// TIA Portal V17 export
// export: Created 2023-12-22T15:05:25.2235005Z, ExportSetting WithDefaults, DisplayName Totally Integrated Automation Portal, DisplayVersion V17, DisplayName TIA Portal Openness, DisplayVersion V17, DisplayName TIA Portal Version Control Interface, DisplayVersion V17, DisplayName STEP 7 Professional, DisplayVersion V17, DisplayName STEP 7 Safety, DisplayVersion V17, DisplayName WinCC Advanced, DisplayVersion V17
FUNCTION_BLOCK "Line_Control"   // FB5, LAD
{ S7_Optimized_Access := 'FALSE' }
VERSION : 0.1
// stored: AutoNumber false, IsIECCheckEnabled false, SetENOAutomatically false, UDAEnableTagReadback false
   VAR DB_SPECIFIC
      Local : Bool;   // Локальный
      RESET_STAT : Bool;   // Обнуление статистики за неделю
      Line_Settings : Bool;   // Параметры линии
      Line_Alarms : Bool;   // Аварии линии
      Group1_PolyMix_1 : Bool;   // Группа 1 PolyMix 1
      Group1_PolyMix_2 : Bool;   // Группа 1 PolyMix 2
      Group2_PolyMix_1 : Bool;   // Группа 2 PolyMix 1
      Group2_PolyMix_2 : Bool;   // Группа 2 PolyMix 2
      ALLS : Bool;   // Нижний аварийный уровень
      REQ_Z6_BK1 : Bool;   // Запрос открытия задвижки 6 с БК 1
      REQ_Z6_BK2 : Bool;   // Запрос открытия задвижки 6 с БК 2
      REQ_Z5_Start_A : Bool;   // Запрос открытия задвижки 5
      REQ_Z4_Start_A : Bool;   // Запрос открытия задвижки 4
      REQ_Z3_Start_A : Bool;   // Запрос открытия задвижки 3
      REQ_Z2_Start_A : Bool;   // Запрос открытия задвижки 2
      REQ_Z1_Start_A : Bool;   // Запрос открытия задвижки 1
      Line_REQ_Settings : Int;   // Запрос параметров линии
      Line_Now_Settings : Int;   // Параметры линии сейчас
      Line_REQ_Alarms : Int;   // Запрос аварий линии
      Line_Now_Alarms : Int;   // Аварии линии сейчас
      All_Lines : Int := 1;   // Кол-во линий
      All_Pumps : Int := 2;   // Кол-во насосов
      Events : Word;   // События
      pos : Array[0..7] of Bool;   // Вспомогательные переменные
   END_VAR
   VAR
      Line { S7_SetPoint := 'True'} : Array[0..2] of "Block_Line";   // Линии (Block Line)
      Pump { S7_SetPoint := 'True'} : Array[1..2] of "Block_Pump";   // Насосы (Block Pump)
   END_VAR
   VAR DB_SPECIFIC
      Time_DTL : DTL;
   END_VAR
   VAR_TEMP
      summ : Real;
      x1 : Bool;
      x2 : Bool;
   END_VAR
   // Line[1].Flow := 1.0;
   // Line[1].LINE_NUMBER := 1;
   // Line[2].LINE_NUMBER := 2;
   // Line[1..2].Hand := true;
   // Line[0].PID.Settings.Max_out := 1.3;
   // Line[0].PID.Settings.Min_out := 0.7;
   // Line[0].PID.Settings.DeadBand := 0.0;
   // Pump[1].PUMP_NUMBER := 1;
   // Pump[2].PUMP_NUMBER := 2;
   // Pump[1].Line_Main := 1;
   // Pump[2].Line_Main := 2;
   VAR_TEMP   // added for the SCL form of the ladder/FBD networks
      _w1 : Bool;
   END_VAR
BEGIN

REGION Network 1: Вызов функций настроек и аварий линий
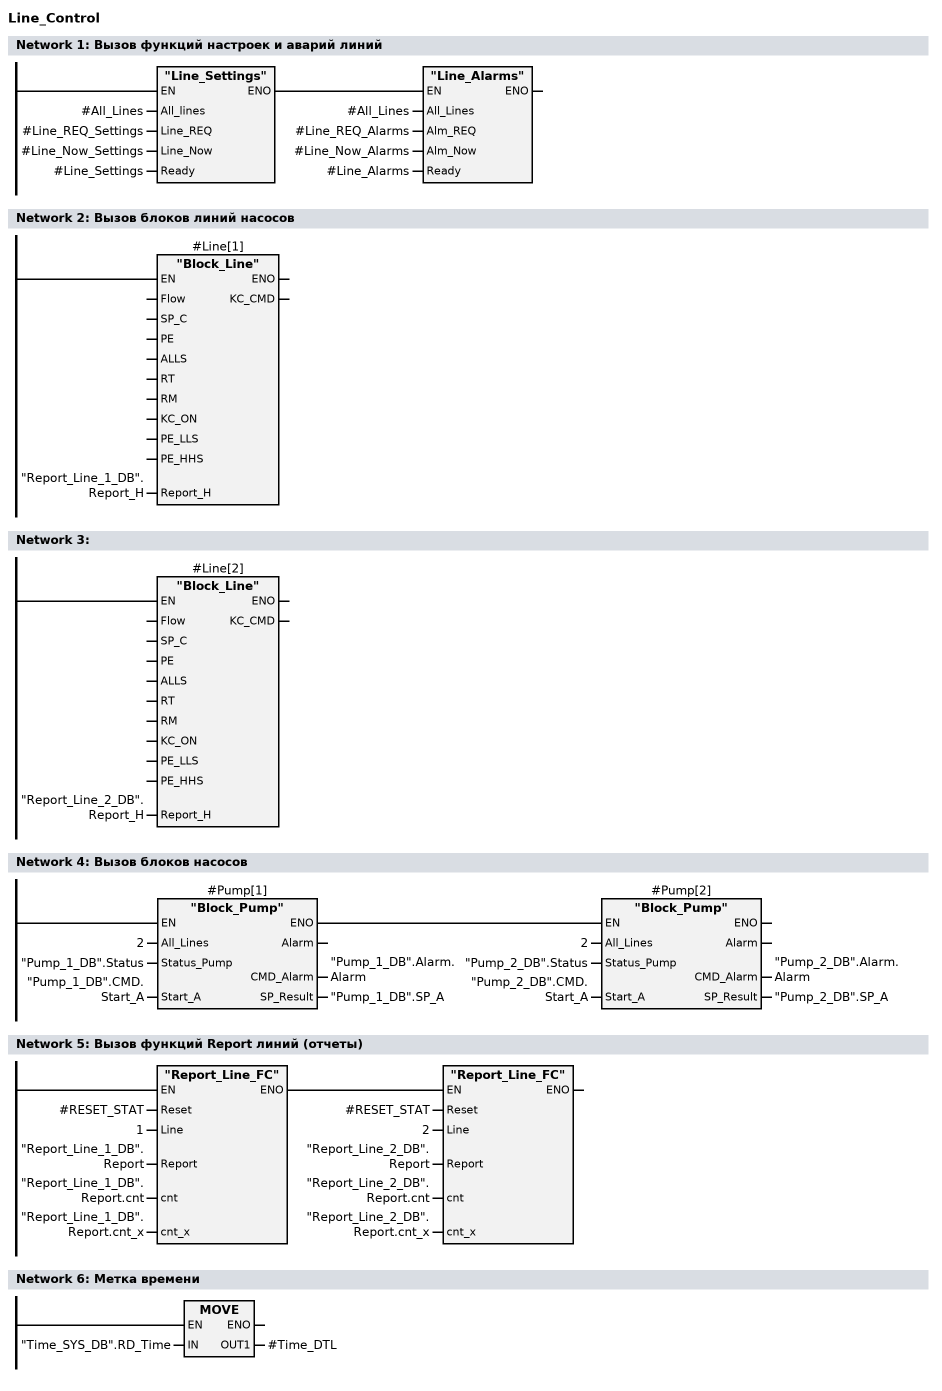
   RUNG wire#powerrail
      "Line_Settings"(All_lines := #All_Lines, Line_REQ := #Line_REQ_Settings, Line_Now := #Line_Now_Settings, Ready := #Line_Settings)
      "Line_Alarms"(All_Lines := #All_Lines, Alm_REQ := #Line_REQ_Alarms, Alm_Now := #Line_Now_Alarms, Ready := #Line_Alarms)
   END_RUNG
   // the same network as SCL:
   "Line_Settings"(All_lines := #All_Lines,
                   Line_REQ := #Line_REQ_Settings,
                   Line_Now := #Line_Now_Settings,
                   Ready := #Line_Settings,
                   ENO => #_w1);
   IF #_w1 THEN
       "Line_Alarms"(All_Lines := #All_Lines,
                     Alm_REQ := #Line_REQ_Alarms,
                     Alm_Now := #Line_Now_Alarms,
                     Ready := #Line_Alarms);
   END_IF;
END_REGION

REGION Network 2: Вызов блоков линий насосов
   RUNG wire#powerrail
      #Line[1](Flow :=, SP_C :=, PE :=, ALLS :=, RT :=, RM :=, KC_ON :=, PE_LLS :=, PE_HHS :=, Report_H := "Report_Line_1_DB".Report_H, KC_CMD =>)
   END_RUNG
   // the same network as SCL:
   #Line[1](Report_H := "Report_Line_1_DB".Report_H);   // "Block_Line"
END_REGION

REGION Network 3
   RUNG wire#powerrail
      #Line[2](Flow :=, SP_C :=, PE :=, ALLS :=, RT :=, RM :=, KC_ON :=, PE_LLS :=, PE_HHS :=, Report_H := "Report_Line_2_DB".Report_H, KC_CMD =>)
   END_RUNG
   // the same network as SCL:
   #Line[2](Report_H := "Report_Line_2_DB".Report_H);   // "Block_Line"
END_REGION

REGION Network 4: Вызов блоков насосов
   RUNG wire#powerrail
      #Pump[1](All_Lines := 2, Status_Pump := "Pump_1_DB".Status, Start_A := "Pump_1_DB".CMD.Start_A, Alarm =>, CMD_Alarm => "Pump_1_DB".Alarm.Alarm, SP_Result => "Pump_1_DB".SP_A)
      #Pump[2](All_Lines := 2, Status_Pump := "Pump_2_DB".Status, Start_A := "Pump_2_DB".CMD.Start_A, Alarm =>, CMD_Alarm => "Pump_2_DB".Alarm.Alarm, SP_Result => "Pump_2_DB".SP_A)
   END_RUNG
   // the same network as SCL:
   #Pump[1](All_Lines := 2,   // "Block_Pump"
            Status_Pump := "Pump_1_DB".Status,
            Start_A := "Pump_1_DB".CMD.Start_A,
            CMD_Alarm => "Pump_1_DB".Alarm.Alarm,
            SP_Result => "Pump_1_DB".SP_A,
            ENO => #_w1);
   IF #_w1 THEN
       #Pump[2](All_Lines := 2,   // "Block_Pump"
                Status_Pump := "Pump_2_DB".Status,
                Start_A := "Pump_2_DB".CMD.Start_A,
                CMD_Alarm => "Pump_2_DB".Alarm.Alarm,
                SP_Result => "Pump_2_DB".SP_A);
   END_IF;
END_REGION

REGION Network 5: Вызов функций Report линий (отчеты)
   RUNG wire#powerrail
      "Report_Line_FC"(Reset := #RESET_STAT, Line := 1, Report := "Report_Line_1_DB".Report, cnt := "Report_Line_1_DB".Report.cnt, cnt_x := "Report_Line_1_DB".Report.cnt_x)
      "Report_Line_FC"(Reset := #RESET_STAT, Line := 2, Report := "Report_Line_2_DB".Report, cnt := "Report_Line_2_DB".Report.cnt, cnt_x := "Report_Line_2_DB".Report.cnt_x)
   END_RUNG
   // the same network as SCL:
   "Report_Line_FC"(Reset := #RESET_STAT,
                    Line := 1,
                    Report := "Report_Line_1_DB".Report,
                    cnt := "Report_Line_1_DB".Report.cnt,
                    cnt_x := "Report_Line_1_DB".Report.cnt_x,
                    ENO => #_w1);
   IF #_w1 THEN
       "Report_Line_FC"(Reset := #RESET_STAT,
                        Line := 2,
                        Report := "Report_Line_2_DB".Report,
                        cnt := "Report_Line_2_DB".Report.cnt,
                        cnt_x := "Report_Line_2_DB".Report.cnt_x);
   END_IF;
END_REGION

REGION Network 6: Метка времени
   RUNG wire#powerrail
      Move(in := "Time_SYS_DB".RD_Time, out1 => #Time_DTL)
   END_RUNG
   // the same network as SCL:
   #Time_DTL := "Time_SYS_DB".RD_Time;
END_REGION
END_FUNCTION_BLOCK
